TYPE csp_transfer_accumulator_belt_cam_enum :
(
	IDLE							:= 33,
	RUN								:= 16	
);
END_TYPE

(* stored: Version 1.1.0.1, ProductVersion 3.1.4022.12
   DUT csp_transfer_accumulator_belt_cam_enum: Id {02407e18-a6d8-405f-bdc2-7e7053b39560} *)
